{attribute wpf [Container(Layout.GroupBox)]}
TYPE GroupBoxLayout:
STRUCT
	{attribute addProperty Name "<#Car - an idea#>"}
	_car: Car;
	
	{attribute addProperty Name "<#An integer#>"}
	_INT_00: INT;
END_STRUCT
END_TYPE

(* stored: Version 1.1.0.1, ProductVersion 3.1.4024.9
   DUT GroupBoxLayout: Id {cad173a1-4b25-44ff-9267-9295204f781a} *)
